LIN {X 0,Y 229.881,Z 707.672,A -85,B 0,C 180,E1 18522.942,E2 18522.942} C_VEL
LIN {X 0,Y 219.787,Z 692.83,A -85,B 0,C 180,E1 18532.814,E2 18532.814} C_VEL
LIN {X 0,Y 216.268,Z 686.361,A -85,B 0,C 180,E1 18540.004,E2 18540.004} C_VEL
LIN {X 0,Y 217.024,Z 688.955,A -85,B 0,C 180,E1 18552.29,E2 18552.29} C_VEL
LIN {X 0,Y 226.193,Z 701.763,A -85,B 0,C 180,E1 18563.446,E2 18563.446} C_VEL
LIN {X 0,Y 243.494,Z 730.82,A -85,B 0,C 180,E1 18574.667,E2 18574.667} C_VEL
LIN {X 0,Y 255.556,Z 766.15,A -85,B 0,C 180,E1 18582.726,E2 18582.726} C_VEL
LIN {X 0,Y 253.616,Z 779.963,A -85,B 0,C 180,E1 18584.484,E2 18584.484} C_VEL
LIN {X 0,Y 237.279,Z 822.45,A -85,B 0,C 180,E1 18590.836,E2 18590.836} C_VEL
LIN {X 0,Y 221.036,Z 856.867,A -85,B 0,C 180,E1 18601.276,E2 18601.276} C_VEL
LIN {X 0,Y 213.518,Z 876.846,A -85,B 0,C 180,E1 18613.662,E2 18613.662} C_VEL
LIN {X 0,Y 213.499,Z 883.891,A -85,B 0,C 180,E1 18623.879,E2 18623.879} C_VEL
LIN {X 0,Y 213.953,Z 882.641,A -85,B 0,C 180,E1 18634.067,E2 18634.067} C_VEL
LIN {X 0,Y 214.175,Z 868.105,A -85,B 0,C 180,E1 18646.928,E2 18646.928} C_VEL
LIN {X 0,Y 220.9,Z 839.18,A -85,B 0,C 180,E1 18658.743,E2 18658.743} C_VEL
LIN {X 0,Y 232.247,Z 798.241,A -85,B 0,C 180,E1 18667.481,E2 18667.481} C_VEL
LIN {X 0,Y 239.047,Z 758.866,A -85,B 0,C 180,E1 18672.107,E2 18672.107} C_VEL
LIN {X 0,Y 223.377,Z 710.425,A -85,B 0,C 180,E1 18677.976,E2 18677.976} C_VEL
LIN {X 0,Y 208.041,Z 678.81,A -85,B 0,C 180,E1 18682.787,E2 18682.787} C_VEL
LIN {X 0,Y 208.536,Z 678.81,A -85,B 0,C 180,E1 18696.401,E2 18696.401} C_VEL
LIN {X 0,Y 209.842,Z 678.81,A -85,B 0,C 180,E1 18709.579,E2 18709.579} C_VEL
LIN {X 0,Y 210.218,Z 678.81,A -85,B 0,C 180,E1 18722.064,E2 18722.064} C_VEL
LIN {X 0,Y 209.548,Z 678.81,A -85,B 0,C 180,E1 18734.679,E2 18734.679} C_VEL
LIN {X 0,Y 208.418,Z 678.81,A -85,B 0,C 180,E1 18748.378,E2 18748.378} C_VEL
LIN {X 0,Y 207.707,Z 678.81,A -85,B 0,C 180,E1 18757.847,E2 18757.847} C_VEL
LIN {X 0,Y 199.525,Z 678.81,A -85,B 0,C 180,E1 18767.645,E2 18767.645} C_VEL
LIN {X 0,Y 200.068,Z 678.81,A -85,B 0,C 180,E1 18780.723,E2 18780.723} C_VEL
LIN {X 0,Y 200.672,Z 680.538,A -85,B 0,C 180,E1 18786.541,E2 18786.541} C_VEL
LIN {X 0,Y 219.908,Z 721.807,A -85,B 0,C 180,E1 18793.945,E2 18793.945} C_VEL
LIN {X 0,Y 225.033,Z 755.949,A -85,B 0,C 180,E1 18800.294,E2 18800.294} C_VEL
LIN {X 0,Y 215.989,Z 790.154,A -85,B 0,C 180,E1 18808.49,E2 18808.49} C_VEL
LIN {X 0,Y 208.94,Z 812.982,A -85,B 0,C 180,E1 18819.406,E2 18819.406} C_VEL
LIN {X 0,Y 206.98,Z 821.875,A -85,B 0,C 180,E1 18829.265,E2 18829.265} C_VEL
LIN {X 0,Y 211.489,Z 820.688,A -85,B 0,C 180,E1 18842.559,E2 18842.559} C_VEL
LIN {X 0,Y 222.679,Z 806.166,A -85,B 0,C 180,E1 18853.748,E2 18853.748} C_VEL
LIN {X 0,Y 239.014,Z 776.963,A -85,B 0,C 180,E1 18862.905,E2 18862.905} C_VEL
LIN {X 0,Y 239.061,Z 749.813,A -85,B 0,C 180,E1 18870.717,E2 18870.717} C_VEL
LIN {X 0,Y 229.457,Z 720.051,A -85,B 0,C 180,E1 18881.194,E2 18881.194} C_VEL
LIN {X 0,Y 218.851,Z 700.999,A -85,B 0,C 180,E1 18892.533,E2 18892.533} C_VEL
LIN {X 0,Y 214.934,Z 694.204,A -85,B 0,C 180,E1 18901.016,E2 18901.016} C_VEL
LIN {X 0,Y 215.807,Z 696.88,A -85,B 0,C 180,E1 18911.921,E2 18911.921} C_VEL
LIN {X 0,Y 224.295,Z 709.472,A -85,B 0,C 180,E1 18922.88,E2 18922.88} C_VEL
LIN {X 0,Y 239.571,Z 737.112,A -85,B 0,C 180,E1 18933.939,E2 18933.939} C_VEL
LIN {X 0,Y 249.788,Z 770.735,A -85,B 0,C 180,E1 18942.009,E2 18942.009} C_VEL
LIN {X 0,Y 234.134,Z 815.138,A -85,B 0,C 180,E1 18948.201,E2 18948.201} C_VEL
LIN {X 0,Y 216.296,Z 851.412,A -85,B 0,C 180,E1 18958.25,E2 18958.25} C_VEL
LIN {X 0,Y 206.081,Z 874.611,A -85,B 0,C 180,E1 18971.855,E2 18971.855} C_VEL
LIN {X 0,Y 205.649,Z 883.042,A -85,B 0,C 180,E1 18985.094,E2 18985.094} C_VEL
LIN {X 0,Y 205.813,Z 879.931,A -85,B 0,C 180,E1 18996.35,E2 18996.35} C_VEL
LIN {X 0,Y 206.758,Z 862.386,A -85,B 0,C 180,E1 19009.844,E2 19009.844} C_VEL
LIN {X 0,Y 215.77,Z 829.843,A -85,B 0,C 180,E1 19021.836,E2 19021.836} C_VEL
LIN {X 0,Y 227.885,Z 786.903,A -85,B 0,C 180,E1 19029.909,E2 19029.909} C_VEL
LIN {X 0,Y 231.839,Z 760.664,A -85,B 0,C 180,E1 19032.91,E2 19032.91} C_VEL
LIN {X 0,Y 217.334,Z 714.047,A -85,B 0,C 180,E1 19038.986,E2 19038.986} C_VEL
LIN {X 0,Y 200.023,Z 678.81,A -85,B 0,C 180,E1 19044.727,E2 19044.727} C_VEL
LIN {X 0,Y 200.91,Z 678.81,A -85,B 0,C 180,E1 19060.764,E2 19060.764} C_VEL
LIN {X 0,Y 202.255,Z 678.81,A -85,B 0,C 180,E1 19073.533,E2 19073.533} C_VEL
LIN {X 0,Y 201.927,Z 678.81,A -85,B 0,C 180,E1 19086.469,E2 19086.469} C_VEL
LIN {X 0,Y 201.016,Z 678.81,A -85,B 0,C 180,E1 19099.856,E2 19099.856} C_VEL
LIN {X 0,Y 199.794,Z 678.81,A -85,B 0,C 180,E1 19114.724,E2 19114.724} C_VEL
LIN {X 0,Y 199.525,Z 678.81,A -85,B 0,C 180,E1 19127.645,E2 19127.645} C_VEL
LIN {X 0,Y 191.668,Z 678.81,A -85,B 0,C 180,E1 19137.868,E2 19137.868} C_VEL
LIN {X 0,Y 192.303,Z 680.013,A -85,B 0,C 180,E1 19144.277,E2 19144.277} C_VEL
LIN {X 0,Y 212.255,Z 721.579,A -85,B 0,C 180,E1 19152.421,E2 19152.421} C_VEL
LIN {X 0,Y 217.81,Z 755.571,A -85,B 0,C 180,E1 19159.042,E2 19159.042} C_VEL
LIN {X 0,Y 208.829,Z 789.974,A -85,B 0,C 180,E1 19167.397,E2 19167.397} C_VEL
LIN {X 0,Y 201.296,Z 813.354,A -85,B 0,C 180,E1 19178.589,E2 19178.589} C_VEL
LIN {X 0,Y 199.104,Z 823.33,A -85,B 0,C 180,E1 19190.059,E2 19190.059} C_VEL
LIN {X 0,Y 204.361,Z 821.543,A -85,B 0,C 180,E1 19203.844,E2 19203.844} C_VEL
LIN {X 0,Y 217.393,Z 805.196,A -85,B 0,C 180,E1 19215.88,E2 19215.88} C_VEL
LIN {X 0,Y 233.806,Z 774.97,A -85,B 0,C 180,E1 19225.119,E2 19225.119} C_VEL
LIN {X 0,Y 232.12,Z 746.503,A -85,B 0,C 180,E1 19234.176,E2 19234.176} C_VEL
LIN {X 0,Y 222.959,Z 720.424,A -85,B 0,C 180,E1 19245.089,E2 19245.089} C_VEL
LIN {X 0,Y 215.766,Z 706.799,A -85,B 0,C 180,E1 19255.213,E2 19255.213} C_VEL
LIN {X 0,Y 213.643,Z 701.951,A -85,B 0,C 180,E1 19262.04,E2 19262.04} C_VEL
LIN {X 0,Y 214.62,Z 705.005,A -85,B 0,C 180,E1 19271.73,E2 19271.73} C_VEL
LIN {X 0,Y 222.354,Z 717.478,A -85,B 0,C 180,E1 19282.508,E2 19282.508} C_VEL
LIN {X 0,Y 235.487,Z 743.318,A -85,B 0,C 180,E1 19293.22,E2 19293.22} C_VEL
LIN {X 0,Y 243.997,Z 775.784,A -85,B 0,C 180,E1 19301.391,E2 19301.391} C_VEL
LIN {X 0,Y 225.894,Z 819.243,A -85,B 0,C 180,E1 19307.758,E2 19307.758} C_VEL
LIN {X 0,Y 207.434,Z 854.096,A -85,B 0,C 180,E1 19318.584,E2 19318.584} C_VEL
LIN {X 0,Y 197.999,Z 874.565,A -85,B 0,C 180,E1 19332.096,E2 19332.096} C_VEL
LIN {X 0,Y 197.523,Z 881.59,A -85,B 0,C 180,E1 19343.382,E2 19343.382} C_VEL
LIN {X 0,Y 197.998,Z 879.68,A -85,B 0,C 180,E1 19354.942,E2 19354.942} C_VEL
LIN {X 0,Y 198.588,Z 863.33,A -85,B 0,C 180,E1 19369.163,E2 19369.163} C_VEL
LIN {X 0,Y 207.077,Z 833.12,A -85,B 0,C 180,E1 19381.476,E2 19381.476} C_VEL
LIN {X 0,Y 219.379,Z 791.904,A -85,B 0,C 180,E1 19390.105,E2 19390.105} C_VEL
LIN {X 0,Y 224.696,Z 762.234,A -85,B 0,C 180,E1 19393.787,E2 19393.787} C_VEL
LIN {X 0,Y 210.704,Z 716.189,A -85,B 0,C 180,E1 19400.235,E2 19400.235} C_VEL
LIN {X 0,Y 191.849,Z 678.81,A -85,B 0,C 180,E1 19406.993,E2 19406.993} C_VEL
LIN {X 0,Y 192.609,Z 678.81,A -85,B 0,C 180,E1 19419.228,E2 19419.228} C_VEL
LIN {X 0,Y 194.175,Z 678.81,A -85,B 0,C 180,E1 19433.263,E2 19433.263} C_VEL
LIN {X 0,Y 193.88,Z 678.81,A -85,B 0,C 180,E1 19446.738,E2 19446.738} C_VEL
LIN {X 0,Y 192.831,Z 678.81,A -85,B 0,C 180,E1 19460.737,E2 19460.737} C_VEL
LIN {X 0,Y 191.686,Z 678.81,A -85,B 0,C 180,E1 19476.421,E2 19476.421} C_VEL
LIN {X 0,Y 191.628,Z 678.81,A -85,B 0,C 180,E1 19493.563,E2 19493.563} C_VEL
LIN {X 0,Y 191.668,Z 678.81,A -85,B 0,C 180,E1 19497.868,E2 19497.868} C_VEL
LIN {X 0,Y 191.635,Z 685.766,A -85,B 0,C 180,E1 19502.561,E2 19502.561} C_VEL
LIN {X 0,Y 194.981,Z 698.935,A -85,B 0,C 180,E1 19506.133,E2 19506.133} C_VEL
LIN {X 0,Y 208.603,Z 735.9,A -85,B 0,C 180,E1 19513.694,E2 19513.694} C_VEL
LIN {X 0,Y 209.864,Z 765.32,A -85,B 0,C 180,E1 19519.915,E2 19519.915} C_VEL
LIN {X 0,Y 199.146,Z 798.07,A -85,B 0,C 180,E1 19529.344,E2 19529.344} C_VEL
LIN {X 0,Y 192.296,Z 818.117,A -85,B 0,C 180,E1 19541.379,E2 19541.379} C_VEL
LIN {X 0,Y 192.318,Z 825.544,A -85,B 0,C 180,E1 19555.721,E2 19555.721} C_VEL
LIN {X 0,Y 201.587,Z 818.107,A -85,B 0,C 180,E1 19569.783,E2 19569.783} C_VEL
LIN {X 0,Y 217.802,Z 796.184,A -85,B 0,C 180,E1 19581.054,E2 19581.054} C_VEL
LIN {X 0,Y 227.781,Z 775.465,A -85,B 0,C 180,E1 19586.917,E2 19586.917} C_VEL
LIN {X 0,Y 226.105,Z 747.296,A -85,B 0,C 180,E1 19596.623,E2 19596.623} C_VEL
LIN {X 0,Y 217.743,Z 722.229,A -85,B 0,C 180,E1 19608.699,E2 19608.699} C_VEL
LIN {X 0,Y 212.516,Z 709.99,A -85,B 0,C 180,E1 19621.027,E2 19621.027} C_VEL
LIN {X 0,Y 213.137,Z 712.726,A -85,B 0,C 180,E1 19631.294,E2 19631.294} C_VEL
LIN {X 0,Y 220.191,Z 725.55,A -85,B 0,C 180,E1 19642.281,E2 19642.281} C_VEL
LIN {X 0,Y 231.93,Z 751.303,A -85,B 0,C 180,E1 19653.122,E2 19653.122} C_VEL
LIN {X 0,Y 237.549,Z 778.975,A -85,B 0,C 180,E1 19660.291,E2 19660.291} C_VEL
LIN {X 0,Y 218.507,Z 821.527,A -85,B 0,C 180,E1 19666.952,E2 19666.952} C_VEL
LIN {X 0,Y 199.834,Z 854.414,A -85,B 0,C 180,E1 19677.887,E2 19677.887} C_VEL
LIN {X 0,Y 190.206,Z 873.601,A -85,B 0,C 180,E1 19691.389,E2 19691.389} C_VEL
LIN {X 0,Y 190.024,Z 880.843,A -85,B 0,C 180,E1 19706.756,E2 19706.756} C_VEL
LIN {X 0,Y 189.875,Z 877.181,A -85,B 0,C 180,E1 19716.885,E2 19716.885} C_VEL
LIN {X 0,Y 191.335,Z 858.875,A -85,B 0,C 180,E1 19731.52,E2 19731.52} C_VEL
LIN {X 0,Y 201.289,Z 827.068,A -85,B 0,C 180,E1 19743.78,E2 19743.78} C_VEL
LIN {X 0,Y 214.537,Z 783.538,A -85,B 0,C 180,E1 19752.221,E2 19752.221} C_VEL
LIN {X 0,Y 217.438,Z 763.356,A -85,B 0,C 180,E1 19754.787,E2 19754.787} C_VEL
LIN {X 0,Y 203.878,Z 717.945,A -85,B 0,C 180,E1 19761.652,E2 19761.652} C_VEL
LIN {X 0,Y 183.912,Z 678.81,A -85,B 0,C 180,E1 19769.058,E2 19769.058} C_VEL
LIN {X 0,Y 184.914,Z 678.81,A -85,B 0,C 180,E1 19783.301,E2 19783.301} C_VEL
LIN {X 0,Y 186.823,Z 678.81,A -85,B 0,C 180,E1 19797.667,E2 19797.667} C_VEL
LIN {X 0,Y 185.641,Z 678.81,A -85,B 0,C 180,E1 19811.788,E2 19811.788} C_VEL
LIN {X 0,Y 184.161,Z 678.81,A -85,B 0,C 180,E1 19826.947,E2 19826.947} C_VEL
LIN {X 0,Y 183.344,Z 678.81,A -85,B 0,C 180,E1 19844.709,E2 19844.709} C_VEL
LIN {X 0,Y 184.123,Z 680.189,A -85,B 0,C 180,E1 19861.813,E2 19861.813} C_VEL
LIN {X 0,Y 194.981,Z 698.935,A -85,B 0,C 180,E1 19866.133,E2 19866.133} C_VEL
LIN {X 0,Y 199.908,Z 730.202,A -85,B 0,C 180,E1 19870.917,E2 19870.917} C_VEL
LIN {X 0,Y 203.53,Z 761.737,A -85,B 0,C 180,E1 19877.89,E2 19877.89} C_VEL
LIN {X 0,Y 192.743,Z 795.512,A -85,B 0,C 180,E1 19887.18,E2 19887.18} C_VEL
LIN {X 0,Y 184.723,Z 818.218,A -85,B 0,C 180,E1 19900.236,E2 19900.236} C_VEL
LIN {X 0,Y 183.458,Z 826.079,A -85,B 0,C 180,E1 19911.854,E2 19911.854} C_VEL
LIN {X 0,Y 190.502,Z 823.157,A -85,B 0,C 180,E1 19926.688,E2 19926.688} C_VEL
LIN {X 0,Y 205.895,Z 805.593,A -85,B 0,C 180,E1 19939.301,E2 19939.301} C_VEL
LIN {X 0,Y 221.461,Z 779.214,A -85,B 0,C 180,E1 19947.714,E2 19947.714} C_VEL
LIN {X 0,Y 221.211,Z 753.146,A -85,B 0,C 180,E1 19957.251,E2 19957.251} C_VEL
LIN {X 0,Y 215.046,Z 729.857,A -85,B 0,C 180,E1 19968.814,E2 19968.814} C_VEL
LIN {X 0,Y 210.827,Z 717.776,A -85,B 0,C 180,E1 19981.035,E2 19981.035} C_VEL
LIN {X 0,Y 211.345,Z 720.576,A -85,B 0,C 180,E1 19991.042,E2 19991.042} C_VEL
LIN {X 0,Y 217.754,Z 733.517,A -85,B 0,C 180,E1 20002.141,E2 20002.141} C_VEL
LIN {X 0,Y 227.73,Z 758.407,A -85,B 0,C 180,E1 20012.79,E2 20012.79} C_VEL
LIN {X 0,Y 231.047,Z 782.48,A -85,B 0,C 180,E1 20019.164,E2 20019.164} C_VEL
LIN {X 0,Y 210.833,Z 824.25,A -85,B 0,C 180,E1 20026.249,E2 20026.249} C_VEL
LIN {X 0,Y 190.974,Z 856.722,A -85,B 0,C 180,E1 20038.234,E2 20038.234} C_VEL
LIN {X 0,Y 181.452,Z 875.348,A -85,B 0,C 180,E1 20054.138,E2 20054.138} C_VEL
LIN {X 0,Y 182.323,Z 879.653,A -85,B 0,C 180,E1 20067.615,E2 20067.615} C_VEL
LIN {X 0,Y 181.577,Z 872.771,A -85,B 0,C 180,E1 20080.839,E2 20080.839} C_VEL
LIN {X 0,Y 185.763,Z 850.113,A -85,B 0,C 180,E1 20096.014,E2 20096.014} C_VEL
LIN {X 0,Y 198.033,Z 814.084,A -85,B 0,C 180,E1 20107.81,E2 20107.81} C_VEL
LIN {X 0,Y 210.974,Z 768.884,A -85,B 0,C 180,E1 20115.096,E2 20115.096} C_VEL
LIN {X 0,Y 198.838,Z 723.531,A -85,B 0,C 180,E1 20122.478,E2 20122.478} C_VEL
LIN {X 0,Y 175.983,Z 678.81,A -85,B 0,C 180,E1 20132.539,E2 20132.539} C_VEL
LIN {X 0,Y 177.584,Z 678.81,A -85,B 0,C 180,E1 20149.337,E2 20149.337} C_VEL
LIN {X 0,Y 178.102,Z 678.81,A -85,B 0,C 180,E1 20162.437,E2 20162.437} C_VEL
LIN {X 0,Y 177.02,Z 678.81,A -85,B 0,C 180,E1 20177.456,E2 20177.456} C_VEL
LIN {X 0,Y 175.448,Z 678.81,A -85,B 0,C 180,E1 20194.744,E2 20194.744} C_VEL
LIN {X 0,Y 175.163,Z 678.81,A -85,B 0,C 180,E1 20209.476,E2 20209.476} C_VEL
LIN {X 0,Y 175.879,Z 680.501,A -85,B 0,C 180,E1 20218.99,E2 20218.99} C_VEL
LIN {X 0,Y 196.233,Z 718.883,A -85,B 0,C 180,E1 20228.459,E2 20228.459} C_VEL
LIN {X 0,Y 199.908,Z 730.202,A -85,B 0,C 180,E1 20230.917,E2 20230.917} C_VEL
LIN {X 0,Y 196.606,Z 760.663,A -85,B 0,C 180,E1 20236.252,E2 20236.252} C_VEL
LIN {X 0,Y 185.716,Z 795.329,A -85,B 0,C 180,E1 20245.9,E2 20245.9} C_VEL
LIN {X 0,Y 176.984,Z 818.89,A -85,B 0,C 180,E1 20259.587,E2 20259.587} C_VEL
LIN {X 0,Y 176.303,Z 827.866,A -85,B 0,C 180,E1 20275.343,E2 20275.343} C_VEL
LIN {X 0,Y 186.15,Z 821.865,A -85,B 0,C 180,E1 20290.703,E2 20290.703} C_VEL
LIN {X 0,Y 204.148,Z 800.993,A -85,B 0,C 180,E1 20303.031,E2 20303.031} C_VEL
LIN {X 0,Y 215.458,Z 781.062,A -85,B 0,C 180,E1 20309.253,E2 20309.253} C_VEL
LIN {X 0,Y 215.942,Z 756.697,A -85,B 0,C 180,E1 20318.839,E2 20318.839} C_VEL
LIN {X 0,Y 211.112,Z 735.388,A -85,B 0,C 180,E1 20330.696,E2 20330.696} C_VEL
LIN {X 0,Y 208.624,Z 725.403,A -85,B 0,C 180,E1 20342.089,E2 20342.089} C_VEL
LIN {X 0,Y 209.224,Z 728.445,A -85,B 0,C 180,E1 20350.928,E2 20350.928} C_VEL
LIN {X 0,Y 214.799,Z 740.892,A -85,B 0,C 180,E1 20361.777,E2 20361.777} C_VEL
LIN {X 0,Y 223.39,Z 766.243,A -85,B 0,C 180,E1 20372.742,E2 20372.742} C_VEL
LIN {X 0,Y 224.629,Z 785.836,A -85,B 0,C 180,E1 20377.998,E2 20377.998} C_VEL
LIN {X 0,Y 203.085,Z 826.997,A -85,B 0,C 180,E1 20385.529,E2 20385.529} C_VEL
LIN {X 0,Y 183.402,Z 856.858,A -85,B 0,C 180,E1 20397.463,E2 20397.463} C_VEL
LIN {X 0,Y 173.541,Z 874.524,A -85,B 0,C 180,E1 20413.836,E2 20413.836} C_VEL
LIN {X 0,Y 174.354,Z 878.411,A -85,B 0,C 180,E1 20427.506,E2 20427.506} C_VEL
LIN {X 0,Y 173.696,Z 872.396,A -85,B 0,C 180,E1 20440.063,E2 20440.063} C_VEL
LIN {X 0,Y 177.216,Z 851.594,A -85,B 0,C 180,E1 20455.496,E2 20455.496} C_VEL
LIN {X 0,Y 189.579,Z 817.024,A -85,B 0,C 180,E1 20467.979,E2 20467.979} C_VEL
LIN {X 0,Y 203.916,Z 771.307,A -85,B 0,C 180,E1 20475.914,E2 20475.914} C_VEL
LIN {X 0,Y 192.92,Z 727.271,A -85,B 0,C 180,E1 20483.663,E2 20483.663} C_VEL
LIN {X 0,Y 170.756,Z 684.849,A -85,B 0,C 180,E1 20493.427,E2 20493.427} C_VEL
LIN {X 0,Y 168.031,Z 678.81,A -85,B 0,C 180,E1 20495.411,E2 20495.411} C_VEL
LIN {X 0,Y 169.908,Z 678.81,A -85,B 0,C 180,E1 20512.295,E2 20512.295} C_VEL
LIN {X 0,Y 170.083,Z 678.81,A -85,B 0,C 180,E1 20522.552,E2 20522.552} C_VEL
LIN {X 0,Y 168.667,Z 678.81,A -85,B 0,C 180,E1 20539.141,E2 20539.141} C_VEL
LIN {X 0,Y 167.217,Z 678.81,A -85,B 0,C 180,E1 20556.145,E2 20556.145} C_VEL
LIN {X 0,Y 167.14,Z 678.81,A -85,B 0,C 180,E1 20573.831,E2 20573.831} C_VEL
LIN {X 0,Y 167.925,Z 681.626,A -85,B 0,C 180,E1 20575.923,E2 20575.923} C_VEL
LIN {X 0,Y 187.694,Z 716.2,A -85,B 0,C 180,E1 20585.858,E2 20585.858} C_VEL
LIN {X 0,Y 196.478,Z 750.492,A -85,B 0,C 180,E1 20593.869,E2 20593.869} C_VEL
LIN {X 0,Y 196.606,Z 760.663,A -85,B 0,C 180,E1 20596.252,E2 20596.252} C_VEL
LIN {X 0,Y 181.741,Z 787.468,A -85,B 0,C 180,E1 20601.78,E2 20601.78} C_VEL
LIN {X 0,Y 170.876,Z 814.989,A -85,B 0,C 180,E1 20615.095,E2 20615.095} C_VEL
LIN {X 0,Y 167.385,Z 826.908,A -85,B 0,C 180,E1 20628.501,E2 20628.501} C_VEL
LIN {X 0,Y 172.888,Z 827.721,A -85,B 0,C 180,E1 20644.788,E2 20644.788} C_VEL
LIN {X 0,Y 187.531,Z 814.98,A -85,B 0,C 180,E1 20658.462,E2 20658.462} C_VEL
LIN {X 0,Y 208.514,Z 787.522,A -85,B 0,C 180,E1 20669.038,E2 20669.038} C_VEL
LIN {X 0,Y 210.916,Z 762.499,A -85,B 0,C 180,E1 20679.47,E2 20679.47} C_VEL
LIN {X 0,Y 207.647,Z 741.923,A -85,B 0,C 180,E1 20691.597,E2 20691.597} C_VEL
LIN {X 0,Y 206.242,Z 733.037,A -85,B 0,C 180,E1 20702.113,E2 20702.113} C_VEL
LIN {X 0,Y 206.72,Z 735.941,A -85,B 0,C 180,E1 20710.58,E2 20710.58} C_VEL
LIN {X 0,Y 212.681,Z 750.912,A -85,B 0,C 180,E1 20723.112,E2 20723.112} C_VEL
LIN {X 0,Y 219.069,Z 776.779,A -85,B 0,C 180,E1 20733.661,E2 20733.661} C_VEL
LIN {X 0,Y 218.631,Z 788.225,A -85,B 0,C 180,E1 20736.661,E2 20736.661} C_VEL
LIN {X 0,Y 196.277,Z 828.113,A -85,B 0,C 180,E1 20744.342,E2 20744.342} C_VEL
LIN {X 0,Y 175.18,Z 857.887,A -85,B 0,C 180,E1 20757.219,E2 20757.219} C_VEL
LIN {X 0,Y 165.466,Z 874.215,A -85,B 0,C 180,E1 20774.395,E2 20774.395} C_VEL
LIN {X 0,Y 166.403,Z 877.163,A -85,B 0,C 180,E1 20787.386,E2 20787.386} C_VEL
LIN {X 0,Y 165.732,Z 870.942,A -85,B 0,C 180,E1 20800.552,E2 20800.552} C_VEL
LIN {X 0,Y 170.234,Z 848.849,A -85,B 0,C 180,E1 20817.132,E2 20817.132} C_VEL
LIN {X 0,Y 183.552,Z 813.223,A -85,B 0,C 180,E1 20829.847,E2 20829.847} C_VEL
LIN {X 0,Y 196.383,Z 769.328,A -85,B 0,C 180,E1 20837.624,E2 20837.624} C_VEL
LIN {X 0,Y 185.101,Z 726.088,A -85,B 0,C 180,E1 20845.861,E2 20845.861} C_VEL
LIN {X 0,Y 163.425,Z 685.316,A -85,B 0,C 180,E1 20856.567,E2 20856.567} C_VEL
LIN {X 0,Y 160.189,Z 678.81,A -85,B 0,C 180,E1 20859.184,E2 20859.184} C_VEL
LIN {X 0,Y 162.627,Z 678.81,A -85,B 0,C 180,E1 20877.32,E2 20877.32} C_VEL
LIN {X 0,Y 161.203,Z 678.81,A -85,B 0,C 180,E1 20893.607,E2 20893.607} C_VEL
LIN {X 0,Y 159.404,Z 678.81,A -85,B 0,C 180,E1 20911.57,E2 20911.57} C_VEL
LIN {X 0,Y 159.077,Z 678.81,A -85,B 0,C 180,E1 20930.803,E2 20930.803} C_VEL
LIN {X 0,Y 180.251,Z 716.053,A -85,B 0,C 180,E1 20943.611,E2 20943.611} C_VEL
LIN {X 0,Y 189.374,Z 750.675,A -85,B 0,C 180,E1 20952.272,E2 20952.272} C_VEL
LIN {X 0,Y 187.091,Z 773.601,A -85,B 0,C 180,E1 20957.919,E2 20957.919} C_VEL
LIN {X 0,Y 181.741,Z 787.468,A -85,B 0,C 180,E1 20961.78,E2 20961.78} C_VEL
LIN {X 0,Y 166.207,Z 808.669,A -85,B 0,C 180,E1 20969.666,E2 20969.666} C_VEL
LIN {X 0,Y 159.577,Z 826.639,A -85,B 0,C 180,E1 20986.041,E2 20986.041} C_VEL
LIN {X 0,Y 162.555,Z 830.166,A -85,B 0,C 180,E1 21000.895,E2 21000.895} C_VEL
LIN {X 0,Y 176.753,Z 820.45,A -85,B 0,C 180,E1 21016.868,E2 21016.868} C_VEL
LIN {X 0,Y 197.463,Z 797.162,A -85,B 0,C 180,E1 21028.337,E2 21028.337} C_VEL
LIN {X 0,Y 203.893,Z 784.648,A -85,B 0,C 180,E1 21032.698,E2 21032.698} C_VEL
LIN {X 0,Y 205.599,Z 762.892,A -85,B 0,C 180,E1 21042.831,E2 21042.831} C_VEL
LIN {X 0,Y 203.597,Z 745.412,A -85,B 0,C 180,E1 21055.294,E2 21055.294} C_VEL
LIN {X 0,Y 203.51,Z 740.566,A -85,B 0,C 180,E1 21062.141,E2 21062.141} C_VEL
LIN {X 0,Y 204.481,Z 745.404,A -85,B 0,C 180,E1 21072.87,E2 21072.87} C_VEL
LIN {X 0,Y 210.18,Z 762.529,A -85,B 0,C 180,E1 21085.146,E2 21085.146} C_VEL
LIN {X 0,Y 213.921,Z 787.913,A -85,B 0,C 180,E1 21094.892,E2 21094.892} C_VEL
LIN {X 0,Y 189.96,Z 828.652,A -85,B 0,C 180,E1 21102.905,E2 21102.905} C_VEL
LIN {X 0,Y 168.365,Z 857.061,A -85,B 0,C 180,E1 21115.713,E2 21115.713} C_VEL
LIN {X 0,Y 157.644,Z 873.134,A -85,B 0,C 180,E1 21133.599,E2 21133.599} C_VEL
LIN {X 0,Y 158.437,Z 875.91,A -85,B 0,C 180,E1 21147.255,E2 21147.255} C_VEL
LIN {X 0,Y 157.773,Z 869.472,A -85,B 0,C 180,E1 21161.091,E2 21161.091} C_VEL
LIN {X 0,Y 163.032,Z 846.606,A -85,B 0,C 180,E1 21178.586,E2 21178.586} C_VEL
LIN {X 0,Y 177.32,Z 810.55,A -85,B 0,C 180,E1 21191.549,E2 21191.549} C_VEL
LIN {X 0,Y 189.271,Z 770.081,A -85,B 0,C 180,E1 21198.924,E2 21198.924} C_VEL
LIN {X 0,Y 178.682,Z 728.066,A -85,B 0,C 180,E1 21207.572,E2 21207.572} C_VEL
LIN {X 0,Y 159.045,Z 690.923,A -85,B 0,C 180,E1 21218.293,E2 21218.293} C_VEL
LIN {X 0,Y 152.534,Z 678.81,A -85,B 0,C 180,E1 21223.511,E2 21223.511} C_VEL
LIN {X 0,Y 154.552,Z 678.81,A -85,B 0,C 180,E1 21237.18,E2 21237.18} C_VEL
LIN {X 0,Y 153.015,Z 678.81,A -85,B 0,C 180,E1 21254.351,E2 21254.351} C_VEL
LIN {X 0,Y 151.206,Z 678.81,A -85,B 0,C 180,E1 21273.499,E2 21273.499} C_VEL
LIN {X 0,Y 151.189,Z 680.403,A -85,B 0,C 180,E1 21287.079,E2 21287.079} C_VEL
LIN {X 0,Y 171.8,Z 713.859,A -85,B 0,C 180,E1 21300.414,E2 21300.414} C_VEL
LIN {X 0,Y 181.997,Z 747.748,A -85,B 0,C 180,E1 21309.765,E2 21309.765} C_VEL
LIN {X 0,Y 180.729,Z 773.086,A -85,B 0,C 180,E1 21316.34,E2 21316.34} C_VEL
LIN {X 0,Y 168.083,Z 804.5,A -85,B 0,C 180,E1 21327.413,E2 21327.413} C_VEL
LIN {X 0,Y 166.207,Z 808.669,A -85,B 0,C 180,E1 21329.666,E2 21329.666} C_VEL
LIN {X 0,Y 152.821,Z 823.544,A -85,B 0,C 180,E1 21340.231,E2 21340.231} C_VEL
LIN {X 0,Y 152.821,Z 831.345,A -85,B 0,C 180,E1 21356.543,E2 21356.543} C_VEL
LIN {X 0,Y 164.559,Z 826.216,A -85,B 0,C 180,E1 21373.761,E2 21373.761} C_VEL
LIN {X 0,Y 185.302,Z 806.737,A -85,B 0,C 180,E1 21387.081,E2 21387.081} C_VEL
LIN {X 0,Y 197.267,Z 790.25,A -85,B 0,C 180,E1 21392.88,E2 21392.88} C_VEL
LIN {X 0,Y 200.645,Z 768.73,A -85,B 0,C 180,E1 21403.486,E2 21403.486} C_VEL
LIN {X 0,Y 200.057,Z 752.488,A -85,B 0,C 180,E1 21415.654,E2 21415.654} C_VEL
LIN {X 0,Y 200.429,Z 747.98,A -85,B 0,C 180,E1 21422.174,E2 21422.174} C_VEL
LIN {X 0,Y 201.771,Z 753.777,A -85,B 0,C 180,E1 21434.154,E2 21434.154} C_VEL
LIN {X 0,Y 206.595,Z 773.47,A -85,B 0,C 180,E1 21446.786,E2 21446.786} C_VEL
LIN {X 0,Y 206.872,Z 792.921,A -85,B 0,C 180,E1 21453.782,E2 21453.782} C_VEL
LIN {X 0,Y 181.428,Z 832.205,A -85,B 0,C 180,E1 21462.358,E2 21462.358} C_VEL
LIN {X 0,Y 158.801,Z 859.577,A -85,B 0,C 180,E1 21476.668,E2 21476.668} C_VEL
LIN {X 0,Y 149.46,Z 873.058,A -85,B 0,C 180,E1 21495.295,E2 21495.295} C_VEL
LIN {X 0,Y 150.471,Z 874.655,A -85,B 0,C 180,E1 21507.109,E2 21507.109} C_VEL
LIN {X 0,Y 149.828,Z 867.952,A -85,B 0,C 180,E1 21521.687,E2 21521.687} C_VEL
LIN {X 0,Y 155.386,Z 845.782,A -85,B 0,C 180,E1 21539.409,E2 21539.409} C_VEL
LIN {X 0,Y 170.294,Z 810.093,A -85,B 0,C 180,E1 21552.803,E2 21552.803} C_VEL
LIN {X 0,Y 182.334,Z 771.872,A -85,B 0,C 180,E1 21560.099,E2 21560.099} C_VEL
LIN {X 0,Y 172.489,Z 730.313,A -85,B 0,C 180,E1 21569.351,E2 21569.351} C_VEL
LIN {X 0,Y 152.994,Z 692.468,A -85,B 0,C 180,E1 21581.467,E2 21581.467} C_VEL
LIN {X 0,Y 145.199,Z 678.81,A -85,B 0,C 180,E1 21589.454,E2 21589.454} C_VEL
LIN {X 0,Y 145.952,Z 678.81,A -85,B 0,C 180,E1 21602.974,E2 21602.974} C_VEL
LIN {X 0,Y 144.067,Z 678.81,A -85,B 0,C 180,E1 21621.629,E2 21621.629} C_VEL
LIN {X 0,Y 143.061,Z 680.494,A -85,B 0,C 180,E1 21640.964,E2 21640.964} C_VEL
LIN {X 0,Y 162.247,Z 709.493,A -85,B 0,C 180,E1 21655.977,E2 21655.977} C_VEL
LIN {X 0,Y 174.073,Z 742.255,A -85,B 0,C 180,E1 21666.254,E2 21666.254} C_VEL
LIN {X 0,Y 175.196,Z 770.457,A -85,B 0,C 180,E1 21674.184,E2 21674.184} C_VEL
LIN {X 0,Y 161.606,Z 803.161,A -85,B 0,C 180,E1 21685.287,E2 21685.287} C_VEL
LIN {X 0,Y 152.821,Z 823.544,A -85,B 0,C 180,E1 21700.231,E2 21700.231} C_VEL
LIN {X 0,Y 144.011,Z 831.623,A -85,B 0,C 180,E1 21713.154,E2 21713.154} C_VEL
LIN {X 0,Y 152.68,Z 830.514,A -85,B 0,C 180,E1 21730.246,E2 21730.246} C_VEL
LIN {X 0,Y 171.92,Z 815.958,A -85,B 0,C 180,E1 21744.991,E2 21744.991} C_VEL
LIN {X 0,Y 191.227,Z 793.462,A -85,B 0,C 180,E1 21754.125,E2 21754.125} C_VEL
LIN {X 0,Y 195.65,Z 772.677,A -85,B 0,C 180,E1 21765.289,E2 21765.289} C_VEL
LIN {X 0,Y 196.344,Z 758.051,A -85,B 0,C 180,E1 21777.907,E2 21777.907} C_VEL
LIN {X 0,Y 197.26,Z 755.646,A -85,B 0,C 180,E1 21786.631,E2 21786.631} C_VEL
LIN {X 0,Y 199.737,Z 768.389,A -85,B 0,C 180,E1 21799.998,E2 21799.998} C_VEL
LIN {X 0,Y 202.27,Z 790.567,A -85,B 0,C 180,E1 21810.91,E2 21810.91} C_VEL
LIN {X 0,Y 197.43,Z 801.444,A -85,B 0,C 180,E1 21813.194,E2 21813.194} C_VEL
LIN {X 0,Y 170.648,Z 838.153,A -85,B 0,C 180,E1 21822.806,E2 21822.806} C_VEL
LIN {X 0,Y 148.068,Z 862.94,A -85,B 0,C 180,E1 21839.176,E2 21839.176} C_VEL
LIN {X 0,Y 141.533,Z 873.314,A -85,B 0,C 180,E1 21860.745,E2 21860.745} C_VEL
LIN {X 0,Y 142.668,Z 871.882,A -85,B 0,C 180,E1 21873.048,E2 21873.048} C_VEL
LIN {X 0,Y 143.315,Z 857.279,A -85,B 0,C 180,E1 21891.753,E2 21891.753} C_VEL
LIN {X 0,Y 155.541,Z 827.55,A -85,B 0,C 180,E1 21908.461,E2 21908.461} C_VEL
LIN {X 0,Y 172.339,Z 786.587,A -85,B 0,C 180,E1 21919.077,E2 21919.077} C_VEL
LIN {X 0,Y 175.133,Z 770.417,A -85,B 0,C 180,E1 21922.081,E2 21922.081} C_VEL
LIN {X 0,Y 165.307,Z 729.682,A -85,B 0,C 180,E1 21932.012,E2 21932.012} C_VEL
LIN {X 0,Y 147.928,Z 696.603,A -85,B 0,C 180,E1 21944.286,E2 21944.286} C_VEL
LIN {X 0,Y 138.131,Z 678.81,A -85,B 0,C 180,E1 21955.625,E2 21955.625} C_VEL
LIN {X 0,Y 137.322,Z 678.81,A -85,B 0,C 180,E1 21969.536,E2 21969.536} C_VEL
LIN {X 0,Y 135.85,Z 678.81,A -85,B 0,C 180,E1 21983.01,E2 21983.01} C_VEL
LIN {X 0,Y 135.146,Z 680.994,A -85,B 0,C 180,E1 21992.296,E2 21992.296} C_VEL
LIN {X 0,Y 145.957,Z 695.503,A -85,B 0,C 180,E1 22005.025,E2 22005.025} C_VEL
LIN {X 0,Y 161.762,Z 724.396,A -85,B 0,C 180,E1 22018.152,E2 22018.152} C_VEL
LIN {X 0,Y 169.174,Z 757.49,A -85,B 0,C 180,E1 22028.577,E2 22028.577} C_VEL
LIN {X 0,Y 165.6,Z 778.62,A -85,B 0,C 180,E1 22034.601,E2 22034.601} C_VEL
LIN {X 0,Y 151.321,Z 810.155,A -85,B 0,C 180,E1 22047.657,E2 22047.657} C_VEL
LIN {X 0,Y 143.779,Z 828.4,A -85,B 0,C 180,E1 22065.3,E2 22065.3} C_VEL
LIN {X 0,Y 144.011,Z 831.623,A -85,B 0,C 180,E1 22073.154,E2 22073.154} C_VEL
LIN {X 0,Y 142.125,Z 833.111,A -85,B 0,C 180,E1 22087.317,E2 22087.317} C_VEL
LIN {X 0,Y 160.385,Z 822.127,A -85,B 0,C 180,E1 22103.539,E2 22103.539} C_VEL
LIN {X 0,Y 185.34,Z 796.539,A -85,B 0,C 180,E1 22115.508,E2 22115.508} C_VEL
LIN {X 0,Y 190.553,Z 778.091,A -85,B 0,C 180,E1 22126.153,E2 22126.153} C_VEL
LIN {X 0,Y 192.337,Z 765.099,A -85,B 0,C 180,E1 22137.964,E2 22137.964} C_VEL
LIN {X 0,Y 193.505,Z 762.952,A -85,B 0,C 180,E1 22146.761,E2 22146.761} C_VEL
LIN {X 0,Y 195.503,Z 776.144,A -85,B 0,C 180,E1 22160.451,E2 22160.451} C_VEL
LIN {X 0,Y 196.439,Z 795.416,A -85,B 0,C 180,E1 22170.149,E2 22170.149} C_VEL
LIN {X 0,Y 168.637,Z 833.716,A -85,B 0,C 180,E1 22179.254,E2 22179.254} C_VEL
LIN {X 0,Y 143.82,Z 859.29,A -85,B 0,C 180,E1 22194.525,E2 22194.525} C_VEL
LIN {X 0,Y 133.618,Z 871.152,A -85,B 0,C 180,E1 22214.915,E2 22214.915} C_VEL
LIN {X 0,Y 134.512,Z 872.138,A -85,B 0,C 180,E1 22226.766,E2 22226.766} C_VEL
LIN {X 0,Y 133.963,Z 866.159,A -85,B 0,C 180,E1 22241.351,E2 22241.351} C_VEL
LIN {X 0,Y 139.971,Z 844.645,A -85,B 0,C 180,E1 22260.996,E2 22260.996} C_VEL
LIN {X 0,Y 156.536,Z 809.035,A -85,B 0,C 180,E1 22275.641,E2 22275.641} C_VEL
LIN {X 0,Y 168.54,Z 774.571,A -85,B 0,C 180,E1 22282.872,E2 22282.872} C_VEL
LIN {X 0,Y 160.422,Z 735.105,A -85,B 0,C 180,E1 22293.191,E2 22293.191} C_VEL
LIN {X 0,Y 144.906,Z 702.967,A -85,B 0,C 180,E1 22305.784,E2 22305.784} C_VEL
LIN {X 0,Y 134.295,Z 685.851,A -85,B 0,C 180,E1 22318.779,E2 22318.779} C_VEL
LIN {X 0,Y 129.401,Z 682.834,A -85,B 0,C 180,E1 22337.718,E2 22337.718} C_VEL
LIN {X 0,Y 133.708,Z 689.308,A -85,B 0,C 180,E1 22351.792,E2 22351.792} C_VEL
LIN {X 0,Y 144.426,Z 704.606,A -85,B 0,C 180,E1 22365.129,E2 22365.129} C_VEL
LIN {X 0,Y 157.645,Z 732.523,A -85,B 0,C 180,E1 22378.032,E2 22378.032} C_VEL
LIN {X 0,Y 162.683,Z 763.246,A -85,B 0,C 180,E1 22388.3,E2 22388.3} C_VEL
LIN {X 0,Y 157.089,Z 783.598,A -85,B 0,C 180,E1 22394.296,E2 22394.296} C_VEL
LIN {X 0,Y 142.385,Z 813.85,A -85,B 0,C 180,E1 22408.473,E2 22408.473} C_VEL
LIN {X 0,Y 135.761,Z 830.019,A -85,B 0,C 180,E1 22426.228,E2 22426.228} C_VEL
LIN {X 0,Y 142.125,Z 833.111,A -85,B 0,C 180,E1 22447.317,E2 22447.317} C_VEL
LIN {X 0,Y 147.733,Z 828.065,A -85,B 0,C 180,E1 22461.052,E2 22461.052} C_VEL
LIN {X 0,Y 173.484,Z 806.626,A -85,B 0,C 180,E1 22474.377,E2 22474.377} C_VEL
LIN {X 0,Y 180.773,Z 796.963,A -85,B 0,C 180,E1 22478.457,E2 22478.457} C_VEL
LIN {X 0,Y 186.256,Z 779.575,A -85,B 0,C 180,E1 22489.996,E2 22489.996} C_VEL
LIN {X 0,Y 189.153,Z 769.368,A -85,B 0,C 180,E1 22502.304,E2 22502.304} C_VEL
LIN {X 0,Y 189.841,Z 775.111,A -85,B 0,C 180,E1 22513.881,E2 22513.881} C_VEL
LIN {X 0,Y 191.041,Z 792.635,A -85,B 0,C 180,E1 22525.913,E2 22525.913} C_VEL
LIN {X 0,Y 189.03,Z 801.13,A -85,B 0,C 180,E1 22529.128,E2 22529.128} C_VEL
LIN {X 0,Y 160.021,Z 836.922,A -85,B 0,C 180,E1 22538.52,E2 22538.52} C_VEL
LIN {X 0,Y 134.237,Z 861.078,A -85,B 0,C 180,E1 22555.58,E2 22555.58} C_VEL
LIN {X 0,Y 125.567,Z 870.916,A -85,B 0,C 180,E1 22579.555,E2 22579.555} C_VEL
LIN {X 0,Y 126.728,Z 869.17,A -85,B 0,C 180,E1 22593.432,E2 22593.432} C_VEL
LIN {X 0,Y 128.12,Z 853.717,A -85,B 0,C 180,E1 22614.492,E2 22614.492} C_VEL
LIN {X 0,Y 141.893,Z 824.79,A -85,B 0,C 180,E1 22631.785,E2 22631.785} C_VEL
LIN {X 0,Y 160.496,Z 783.437,A -85,B 0,C 180,E1 22642.792,E2 22642.792} C_VEL
LIN {X 0,Y 159.44,Z 756.765,A -85,B 0,C 180,E1 22649.618,E2 22649.618} C_VEL
LIN {X 0,Y 148.376,Z 721.743,A -85,B 0,C 180,E1 22661.16,E2 22661.16} C_VEL
LIN {X 0,Y 134.895,Z 697.201,A -85,B 0,C 180,E1 22675.915,E2 22675.915} C_VEL
LIN {X 0,Y 129.387,Z 690.853,A -85,B 0,C 180,E1 22687.75,E2 22687.75} C_VEL
LIN {X 0,Y 131.392,Z 694.581,A -85,B 0,C 180,E1 22709.033,E2 22709.033} C_VEL
LIN {X 0,Y 142.959,Z 714.496,A -85,B 0,C 180,E1 22725.858,E2 22725.858} C_VEL
LIN {X 0,Y 153.559,Z 742.137,A -85,B 0,C 180,E1 22738.568,E2 22738.568} C_VEL
LIN {X 0,Y 155.709,Z 771.121,A -85,B 0,C 180,E1 22748.755,E2 22748.755} C_VEL
LIN {X 0,Y 139.688,Z 805.929,A -85,B 0,C 180,E1 22761.729,E2 22761.729} C_VEL
LIN {X 0,Y 128.871,Z 827.454,A -85,B 0,C 180,E1 22780.174,E2 22780.174} C_VEL
LIN {X 0,Y 130.697,Z 835.081,A -85,B 0,C 180,E1 22801.501,E2 22801.501} C_VEL
LIN {X 0,Y 147.733,Z 828.065,A -85,B 0,C 180,E1 22821.052,E2 22821.052} C_VEL
LIN {X 0,Y 159.407,Z 816.535,A -85,B 0,C 180,E1 22832.794,E2 22832.794} C_VEL
LIN {X 0,Y 174.264,Z 801.733,A -85,B 0,C 180,E1 22839.038,E2 22839.038} C_VEL
LIN {X 0,Y 180.922,Z 785.873,A -85,B 0,C 180,E1 22850.201,E2 22850.201} C_VEL
LIN {X 0,Y 184.731,Z 776.169,A -85,B 0,C 180,E1 22862.359,E2 22862.359} C_VEL
LIN {X 0,Y 185.254,Z 782.246,A -85,B 0,C 180,E1 22874.232,E2 22874.232} C_VEL
LIN {X 0,Y 185.265,Z 798.906,A -85,B 0,C 180,E1 22885.794,E2 22885.794} C_VEL
LIN {X 0,Y 180.531,Z 807.439,A -85,B 0,C 180,E1 22888.038,E2 22888.038} C_VEL
LIN {X 0,Y 149.968,Z 841.165,A -85,B 0,C 180,E1 22898.39,E2 22898.39} C_VEL
LIN {X 0,Y 124.72,Z 862.458,A -85,B 0,C 180,E1 22916.801,E2 22916.801} C_VEL
LIN {X 0,Y 117.601,Z 869.682,A -85,B 0,C 180,E1 22938.839,E2 22938.839} C_VEL
LIN {X 0,Y 118.742,Z 867.802,A -85,B 0,C 180,E1 22953.663,E2 22953.663} C_VEL
LIN {X 0,Y 120.626,Z 851.915,A -85,B 0,C 180,E1 22976.124,E2 22976.124} C_VEL
LIN {X 0,Y 136.137,Z 821.681,A -85,B 0,C 180,E1 22994.385,E2 22994.385} C_VEL
LIN {X 0,Y 155.185,Z 780.949,A -85,B 0,C 180,E1 23005.016,E2 23005.016} C_VEL
LIN {X 0,Y 149.764,Z 743.341,A -85,B 0,C 180,E1 23016.478,E2 23016.478} C_VEL
LIN {X 0,Y 137.626,Z 712.857,A -85,B 0,C 180,E1 23030.473,E2 23030.473} C_VEL
LIN {X 0,Y 130.389,Z 700.687,A -85,B 0,C 180,E1 23042.182,E2 23042.182} C_VEL
LIN {X 0,Y 127.47,Z 699.263,A -85,B 0,C 180,E1 23059.06,E2 23059.06} C_VEL
LIN {X 0,Y 131.557,Z 706.679,A -85,B 0,C 180,E1 23072.481,E2 23072.481} C_VEL
LIN {X 0,Y 140.905,Z 724.13,A -85,B 0,C 180,E1 23086.588,E2 23086.588} C_VEL
LIN {X 0,Y 148.75,Z 751.824,A -85,B 0,C 180,E1 23099.284,E2 23099.284} C_VEL
LIN {X 0,Y 147.726,Z 777.458,A -85,B 0,C 180,E1 23108.584,E2 23108.584} C_VEL
LIN {X 0,Y 130.373,Z 810.63,A -85,B 0,C 180,E1 23122.639,E2 23122.639} C_VEL
LIN {X 0,Y 120.307,Z 830.316,A -85,B 0,C 180,E1 23142.71,E2 23142.71} C_VEL
LIN {X 0,Y 123.584,Z 836.288,A -85,B 0,C 180,E1 23163.544,E2 23163.544} C_VEL
LIN {X 0,Y 141.965,Z 829.107,A -85,B 0,C 180,E1 23183.295,E2 23183.295} C_VEL
LIN {X 0,Y 159.407,Z 816.535,A -85,B 0,C 180,E1 23192.794,E2 23192.794} C_VEL
LIN {X 0,Y 167.631,Z 806.196,A -85,B 0,C 180,E1 23199.821,E2 23199.821} C_VEL
LIN {X 0,Y 175.735,Z 790.935,A -85,B 0,C 180,E1 23211.315,E2 23211.315} C_VEL
LIN {X 0,Y 180.006,Z 782.754,A -85,B 0,C 180,E1 23222.421,E2 23222.421} C_VEL
LIN {X 0,Y 180.309,Z 789.132,A -85,B 0,C 180,E1 23234.56,E2 23234.56} C_VEL
LIN {X 0,Y 178.828,Z 804.694,A -85,B 0,C 180,E1 23245.313,E2 23245.313} C_VEL
LIN {X 0,Y 148.112,Z 837.849,A -85,B 0,C 180,E1 23254.57,E2 23254.57} C_VEL
LIN {X 0,Y 119.446,Z 860.387,A -85,B 0,C 180,E1 23272.88,E2 23272.88} C_VEL
LIN {X 0,Y 109.653,Z 868.448,A -85,B 0,C 180,E1 23298.018,E2 23298.018} C_VEL
LIN {X 0,Y 110.767,Z 866.429,A -85,B 0,C 180,E1 23313.928,E2 23313.928} C_VEL
LIN {X 0,Y 113.298,Z 850.115,A -85,B 0,C 180,E1 23337.956,E2 23337.956} C_VEL
LIN {X 0,Y 129.963,Z 819.819,A -85,B 0,C 180,E1 23356.672,E2 23356.672} C_VEL
LIN {X 0,Y 148.538,Z 780.477,A -85,B 0,C 180,E1 23367.272,E2 23367.272} C_VEL
LIN {X 0,Y 143.885,Z 745.031,A -85,B 0,C 180,E1 23379.14,E2 23379.14} C_VEL
LIN {X 0,Y 133.578,Z 717.379,A -85,B 0,C 180,E1 23393.587,E2 23393.587} C_VEL
LIN {X 0,Y 128.403,Z 707.902,A -85,B 0,C 180,E1 23404.125,E2 23404.125} C_VEL
LIN {X 0,Y 126.528,Z 707.851,A -85,B 0,C 180,E1 23421.279,E2 23421.279} C_VEL
LIN {X 0,Y 131.754,Z 718.459,A -85,B 0,C 180,E1 23436.444,E2 23436.444} C_VEL
LIN {X 0,Y 140.713,Z 742.688,A -85,B 0,C 180,E1 23452.014,E2 23452.014} C_VEL
LIN {X 0,Y 143.054,Z 770.921,A -85,B 0,C 180,E1 23463.942,E2 23463.942} C_VEL
LIN {X 0,Y 134.289,Z 791.93,A -85,B 0,C 180,E1 23471.039,E2 23471.039} C_VEL
LIN {X 0,Y 117.836,Z 820.294,A -85,B 0,C 180,E1 23488.155,E2 23488.155} C_VEL
LIN {X 0,Y 111.958,Z 834.671,A -85,B 0,C 180,E1 23509.808,E2 23509.808} C_VEL
LIN {X 0,Y 121.825,Z 836.59,A -85,B 0,C 180,E1 23533.245,E2 23533.245} C_VEL
LIN {X 0,Y 146.707,Z 823.714,A -85,B 0,C 180,E1 23551.552,E2 23551.552} C_VEL
LIN {X 0,Y 167.631,Z 806.196,A -85,B 0,C 180,E1 23559.821,E2 23559.821} C_VEL
LIN {X 0,Y 169.942,Z 796.818,A -85,B 0,C 180,E1 23571.575,E2 23571.575} C_VEL
LIN {X 0,Y 174.973,Z 789.129,A -85,B 0,C 180,E1 23582.491,E2 23582.491} C_VEL
LIN {X 0,Y 174.995,Z 795.908,A -85,B 0,C 180,E1 23595.012,E2 23595.012} C_VEL
LIN {X 0,Y 172.639,Z 808.009,A -85,B 0,C 180,E1 23603.531,E2 23603.531} C_VEL
LIN {X 0,Y 139.445,Z 840.708,A -85,B 0,C 180,E1 23613.566,E2 23613.566} C_VEL
LIN {X 0,Y 111.345,Z 860.523,A -85,B 0,C 180,E1 23632.17,E2 23632.17} C_VEL
LIN {X 0,Y 101.722,Z 867.212,A -85,B 0,C 180,E1 23657.069,E2 23657.069} C_VEL
LIN {X 0,Y 102.767,Z 865.011,A -85,B 0,C 180,E1 23674.234,E2 23674.234} C_VEL
LIN {X 0,Y 106.11,Z 848.228,A -85,B 0,C 180,E1 23700.037,E2 23700.037} C_VEL
LIN {X 0,Y 124.813,Z 816.698,A -85,B 0,C 180,E1 23719.649,E2 23719.649} C_VEL
LIN {X 0,Y 142.002,Z 780.906,A -85,B 0,C 180,E1 23729.485,E2 23729.485} C_VEL
LIN {X 0,Y 137.94,Z 746.052,A -85,B 0,C 180,E1 23742.382,E2 23742.382} C_VEL
LIN {X 0,Y 129.509,Z 720.664,A -85,B 0,C 180,E1 23757.685,E2 23757.685} C_VEL
LIN {X 0,Y 125.308,Z 713.851,A -85,B 0,C 180,E1 23770.46,E2 23770.46} C_VEL
LIN {X 0,Y 126.574,Z 720.438,A -85,B 0,C 180,E1 23789.278,E2 23789.278} C_VEL
LIN {X 0,Y 132.996,Z 737.174,A -85,B 0,C 180,E1 23804.464,E2 23804.464} C_VEL
LIN {X 0,Y 137.187,Z 762.798,A -85,B 0,C 180,E1 23817.628,E2 23817.628} C_VEL
LIN {X 0,Y 134.157,Z 781.592,A -85,B 0,C 180,E1 23825.172,E2 23825.172} C_VEL
LIN {X 0,Y 115.568,Z 813.17,A -85,B 0,C 180,E1 23839.983,E2 23839.983} C_VEL
LIN {X 0,Y 104.417,Z 832.617,A -85,B 0,C 180,E1 23862.592,E2 23862.592} C_VEL
LIN {X 0,Y 109.938,Z 838.675,A -85,B 0,C 180,E1 23888.401,E2 23888.401} C_VEL
LIN {X 0,Y 132.524,Z 830.503,A -85,B 0,C 180,E1 23909.186,E2 23909.186} C_VEL
LIN {X 0,Y 162.82,Z 808.125,A -85,B 0,C 180,E1 23922.246,E2 23922.246} C_VEL
LIN {X 0,Y 169.942,Z 796.818,A -85,B 0,C 180,E1 23931.575,E2 23931.575} C_VEL
LIN {X 0,Y 169.963,Z 794.799,A -85,B 0,C 180,E1 23940.581,E2 23940.581} C_VEL
LIN {X 0,Y 169.577,Z 795.553,A -85,B 0,C 180,E1 23943.676,E2 23943.676} C_VEL
LIN {X 0,Y 169.4,Z 801.749,A -85,B 0,C 180,E1 23954.801,E2 23954.801} C_VEL
LIN {X 0,Y 166.77,Z 810.977,A -85,B 0,C 180,E1 23961.605,E2 23961.605} C_VEL
LIN {X 0,Y 131.929,Z 842.393,A -85,B 0,C 180,E1 23971.969,E2 23971.969} C_VEL
LIN {X 0,Y 101.737,Z 861.381,A -85,B 0,C 180,E1 23993.374,E2 23993.374} C_VEL
LIN {X 0,Y 94.529,Z 865.638,A -85,B 0,C 180,E1 24025.396,E2 24025.396} C_VEL
LIN {X 0,Y 94.354,Z 859.555,A -85,B 0,C 180,E1 24043.96,E2 24043.96} C_VEL
LIN {X 0,Y 105.138,Z 836.965,A -85,B 0,C 180,E1 24070.505,E2 24070.505} C_VEL
LIN {X 0,Y 127.331,Z 800.946,A -85,B 0,C 180,E1 24086.89,E2 24086.89} C_VEL
LIN {X 0,Y 135.614,Z 781.991,A -85,B 0,C 180,E1 24091.703,E2 24091.703} C_VEL
LIN {X 0,Y 132.698,Z 748.96,A -85,B 0,C 180,E1 24105.091,E2 24105.091} C_VEL
LIN {X 0,Y 126.052,Z 725.267,A -85,B 0,C 180,E1 24121.382,E2 24121.382} C_VEL
LIN {X 0,Y 122.851,Z 722.382,A -85,B 0,C 180,E1 24137.104,E2 24137.104} C_VEL
LIN {X 0,Y 125.324,Z 731.024,A -85,B 0,C 180,E1 24153.012,E2 24153.012} C_VEL
LIN {X 0,Y 130.531,Z 752.868,A -85,B 0,C 180,E1 24169.079,E2 24169.079} C_VEL
LIN {X 0,Y 129.863,Z 779.228,A -85,B 0,C 180,E1 24181.84,E2 24181.84} C_VEL
LIN {X 0,Y 109.603,Z 812.485,A -85,B 0,C 180,E1 24196.998,E2 24196.998} C_VEL
LIN {X 0,Y 96.668,Z 833.185,A -85,B 0,C 180,E1 24221.317,E2 24221.317} C_VEL
LIN {X 0,Y 103.445,Z 839.813,A -85,B 0,C 180,E1 24251.312,E2 24251.312} C_VEL
LIN {X 0,Y 128.391,Z 831.2,A -85,B 0,C 180,E1 24272.435,E2 24272.435} C_VEL
LIN {X 0,Y 158.215,Z 810.162,A -85,B 0,C 180,E1 24284.866,E2 24284.866} C_VEL
LIN {X 0,Y 165.732,Z 799.906,A -85,B 0,C 180,E1 24294.751,E2 24294.751} C_VEL
LIN {X 0,Y 169.577,Z 795.553,A -85,B 0,C 180,E1 24303.676,E2 24303.676} C_VEL
LIN {X 0,Y 163.409,Z 807.85,A -85,B 0,C 180,E1 24315.11,E2 24315.11} C_VEL
LIN {X 0,Y 160.587,Z 814.321,A -85,B 0,C 180,E1 24319.661,E2 24319.661} C_VEL
LIN {X 0,Y 123.471,Z 844.604,A -85,B 0,C 180,E1 24330.643,E2 24330.643} C_VEL
LIN {X 0,Y 95.27,Z 860.343,A -85,B 0,C 180,E1 24350.419,E2 24350.419} C_VEL
LIN {X 0,Y 86.531,Z 864.309,A -85,B 0,C 180,E1 24384.969,E2 24384.969} C_VEL
LIN {X 0,Y 86.486,Z 857.965,A -85,B 0,C 180,E1 24405.26,E2 24405.26} C_VEL
LIN {X 0,Y 99,Z 834.865,A -85,B 0,C 180,E1 24433.613,E2 24433.613} C_VEL
LIN {X 0,Y 122.564,Z 798.707,A -85,B 0,C 180,E1 24449.891,E2 24449.891} C_VEL
LIN {X 0,Y 129.367,Z 782.751,A -85,B 0,C 180,E1 24454.23,E2 24454.23} C_VEL
LIN {X 0,Y 127.903,Z 753.524,A -85,B 0,C 180,E1 24467.138,E2 24467.138} C_VEL
LIN {X 0,Y 123.5,Z 733.18,A -85,B 0,C 180,E1 24481.753,E2 24481.753} C_VEL
LIN {X 0,Y 121.337,Z 729.396,A -85,B 0,C 180,E1 24490.806,E2 24490.806} C_VEL
LIN {X 0,Y 121.309,Z 735.649,A -85,B 0,C 180,E1 24508.45,E2 24508.45} C_VEL
LIN {X 0,Y 124.902,Z 752.69,A -85,B 0,C 180,E1 24524.24,E2 24524.24} C_VEL
LIN {X 0,Y 124.611,Z 776.634,A -85,B 0,C 180,E1 24537.444,E2 24537.444} C_VEL
LIN {X 0,Y 117.473,Z 791.631,A -85,B 0,C 180,E1 24543.119,E2 24543.119} C_VEL
LIN {X 0,Y 96.559,Z 821.631,A -85,B 0,C 180,E1 24562.096,E2 24562.096} C_VEL
LIN {X 0,Y 88.153,Z 837.309,A -85,B 0,C 180,E1 24588.791,E2 24588.791} C_VEL
LIN {X 0,Y 98.411,Z 840.849,A -85,B 0,C 180,E1 24616.068,E2 24616.068} C_VEL
LIN {X 0,Y 127.253,Z 830.546,A -85,B 0,C 180,E1 24637.098,E2 24637.098} C_VEL
LIN {X 0,Y 153.199,Z 812.897,A -85,B 0,C 180,E1 24647.173,E2 24647.173} C_VEL
LIN {X 0,Y 162.098,Z 802.83,A -85,B 0,C 180,E1 24659.21,E2 24659.21} C_VEL
LIN {X 0,Y 163.97,Z 801.4,A -85,B 0,C 180,E1 24663.47,E2 24663.47} C_VEL
LIN {X 0,Y 163.409,Z 807.85,A -85,B 0,C 180,E1 24675.11,E2 24675.11} C_VEL
LIN {X 0,Y 155.405,Z 816.939,A -85,B 0,C 180,E1 24677.873,E2 24677.873} C_VEL
LIN {X 0,Y 148.086,Z 823.186,A -85,B 0,C 180,E1 24678.902,E2 24678.902} C_VEL
LIN {X 0,Y 110.788,Z 848.936,A -85,B 0,C 180,E1 24691.117,E2 24691.117} C_VEL
LIN {X 0,Y 83.939,Z 861.461,A -85,B 0,C 180,E1 24714.468,E2 24714.468} C_VEL
LIN {X 0,Y 78.711,Z 862.068,A -85,B 0,C 180,E1 24750,E2 24750} C_VEL
LIN {X 0,Y 81.383,Z 849.025,A -85,B 0,C 180,E1 24780.04,E2 24780.04} C_VEL
LIN {X 0,Y 102.279,Z 820.234,A -85,B 0,C 180,E1 24804.691,E2 24804.691} C_VEL
LIN {X 0,Y 123.101,Z 786.031,A -85,B 0,C 180,E1 24815.916,E2 24815.916} C_VEL
LIN {X 0,Y 123.106,Z 757.99,A -85,B 0,C 180,E1 24829.336,E2 24829.336} C_VEL
LIN {X 0,Y 120.353,Z 739.577,A -85,B 0,C 180,E1 24843.607,E2 24843.607} C_VEL
LIN {X 0,Y 117.962,Z 738.172,A -85,B 0,C 180,E1 24858.754,E2 24858.754} C_VEL
LIN {X 0,Y 119.344,Z 750.415,A -85,B 0,C 180,E1 24876.503,E2 24876.503} C_VEL
LIN {X 0,Y 119.814,Z 771.759,A -85,B 0,C 180,E1 24891.131,E2 24891.131} C_VEL
LIN {X 0,Y 115.798,Z 786.252,A -85,B 0,C 180,E1 24898.209,E2 24898.209} C_VEL
LIN {X 0,Y 92.75,Z 818.332,A -85,B 0,C 180,E1 24915.793,E2 24915.793} C_VEL
LIN {X 0,Y 80.235,Z 837.53,A -85,B 0,C 180,E1 24946.482,E2 24946.482} C_VEL
LIN {X 0,Y 91.446,Z 842.09,A -85,B 0,C 180,E1 24978.313,E2 24978.313} C_VEL
LIN {X 0,Y 121.488,Z 832.536,A -85,B 0,C 180,E1 24999.53,E2 24999.53} C_VEL
LIN {X 0,Y 148.265,Z 815.688,A -85,B 0,C 180,E1 25009.579,E2 25009.579} C_VEL
LIN {X 0,Y 156.883,Z 807.744,A -85,B 0,C 180,E1 25020.767,E2 25020.767} C_VEL
LIN {X 0,Y 157.878,Z 810.54,A -85,B 0,C 180,E1 25031.733,E2 25031.733} C_VEL
LIN {X 0,Y 154.857,Z 817.06,A -85,B 0,C 180,E1 25037.492,E2 25037.492} C_VEL
LIN {X 0,Y 148.086,Z 823.186,A -85,B 0,C 180,E1 25038.902,E2 25038.902} C_VEL
LIN {X 0,Y 118.976,Z 841.457,A -85,B 0,C 180,E1 25042.649,E2 25042.649} C_VEL
LIN {X 0,Y 83.273,Z 858.275,A -85,B 0,C 180,E1 25063.201,E2 25063.201} C_VEL
LIN {X 0,Y 70.506,Z 861.639,A -85,B 0,C 180,E1 25103.822,E2 25103.822} C_VEL
LIN {X 0,Y 70.875,Z 854.765,A -85,B 0,C 180,E1 25128.734,E2 25128.734} C_VEL
LIN {X 0,Y 87.772,Z 830.434,A -85,B 0,C 180,E1 25161.081,E2 25161.081} C_VEL
LIN {X 0,Y 114.666,Z 793.15,A -85,B 0,C 180,E1 25176.835,E2 25176.835} C_VEL
LIN {X 0,Y 118.214,Z 777.003,A -85,B 0,C 180,E1 25183.594,E2 25183.594} C_VEL
LIN {X 0,Y 117.719,Z 753.304,A -85,B 0,C 180,E1 25198.146,E2 25198.146} C_VEL
LIN {X 0,Y 116.449,Z 745.36,A -85,B 0,C 180,E1 25207.857,E2 25207.857} C_VEL
LIN {X 0,Y 114.72,Z 748.533,A -85,B 0,C 180,E1 25224.831,E2 25224.831} C_VEL
LIN {X 0,Y 115.244,Z 763.417,A -85,B 0,C 180,E1 25240.945,E2 25240.945} C_VEL
LIN {X 0,Y 111.778,Z 785.228,A -85,B 0,C 180,E1 25254.574,E2 25254.574} C_VEL
LIN {X 0,Y 87.056,Z 818.067,A -85,B 0,C 180,E1 25272.038,E2 25272.038} C_VEL
LIN {X 0,Y 72.663,Z 837.086,A -85,B 0,C 180,E1 25302.055,E2 25302.055} C_VEL
LIN {X 0,Y 78.71,Z 843.363,A -85,B 0,C 180,E1 25332.44,E2 25332.44} C_VEL
LIN {X 0,Y 106.564,Z 838.228,A -85,B 0,C 180,E1 25357.767,E2 25357.767} C_VEL
LIN {X 0,Y 141.947,Z 819.772,A -85,B 0,C 180,E1 25370.778,E2 25370.778} C_VEL
LIN {X 0,Y 151.911,Z 812.304,A -85,B 0,C 180,E1 25382.869,E2 25382.869} C_VEL
LIN {X 0,Y 151.295,Z 816.825,A -85,B 0,C 180,E1 25393.05,E2 25393.05} C_VEL
LIN {X 0,Y 147.641,Z 821.097,A -85,B 0,C 180,E1 25395.502,E2 25395.502} C_VEL
LIN {X 0,Y 118.976,Z 841.457,A -85,B 0,C 180,E1 25402.649,E2 25402.649} C_VEL
LIN {X 0,Y 88.709,Z 853.506,A -85,B 0,C 180,E1 25410.504,E2 25410.504} C_VEL
LIN {X 0,Y 62.779,Z 860.925,A -85,B 0,C 180,E1 25448.74,E2 25448.74} C_VEL
LIN {X 0,Y 62.785,Z 857.761,A -85,B 0,C 180,E1 25476.941,E2 25476.941} C_VEL
LIN {X 0,Y 73.548,Z 838.514,A -85,B 0,C 180,E1 25516.233,E2 25516.233} C_VEL
LIN {X 0,Y 101.231,Z 805.37,A -85,B 0,C 180,E1 25536.662,E2 25536.662} C_VEL
LIN {X 0,Y 111.461,Z 788.594,A -85,B 0,C 180,E1 25541.644,E2 25541.644} C_VEL
LIN {X 0,Y 113.7,Z 763.85,A -85,B 0,C 180,E1 25556.166,E2 25556.166} C_VEL
LIN {X 0,Y 113.19,Z 752.702,A -85,B 0,C 180,E1 25568.085,E2 25568.085} C_VEL
LIN {X 0,Y 111.118,Z 756.05,A -85,B 0,C 180,E1 25584.898,E2 25584.898} C_VEL
LIN {X 0,Y 110.163,Z 770.655,A -85,B 0,C 180,E1 25600.743,E2 25600.743} C_VEL
LIN {X 0,Y 105.09,Z 788.841,A -85,B 0,C 180,E1 25612.141,E2 25612.141} C_VEL
LIN {X 0,Y 79.233,Z 820.31,A -85,B 0,C 180,E1 25630.198,E2 25630.198} C_VEL
LIN {X 0,Y 64.526,Z 838.738,A -85,B 0,C 180,E1 25663.571,E2 25663.571} C_VEL
LIN {X 0,Y 72.719,Z 844.625,A -85,B 0,C 180,E1 25696.921,E2 25696.921} C_VEL
LIN {X 0,Y 103.659,Z 839.025,A -85,B 0,C 180,E1 25722.1,E2 25722.1} C_VEL
LIN {X 0,Y 137.138,Z 822.652,A -85,B 0,C 180,E1 25733.336,E2 25733.336} C_VEL
LIN {X 0,Y 145.431,Z 817.469,A -85,B 0,C 180,E1 25742.997,E2 25742.997} C_VEL
LIN {X 0,Y 145.273,Z 820.295,A -85,B 0,C 180,E1 25750.948,E2 25750.948} C_VEL
LIN {X 0,Y 140.312,Z 824.933,A -85,B 0,C 180,E1 25753.35,E2 25753.35} C_VEL
LIN {X 0,Y 100.167,Z 848.816,A -85,B 0,C 180,E1 25764.63,E2 25764.63} C_VEL
LIN {X 0,Y 88.709,Z 853.506,A -85,B 0,C 180,E1 25770.504,E2 25770.504} C_VEL
LIN {X 0,Y 61.596,Z 858.794,A -85,B 0,C 180,E1 25787.818,E2 25787.818} C_VEL
LIN {X 0,Y 54.999,Z 857.877,A -85,B 0,C 180,E1 25829.999,E2 25829.999} C_VEL
LIN {X 0,Y 63.098,Z 841.63,A -85,B 0,C 180,E1 25874.529,E2 25874.529} C_VEL
LIN {X 0,Y 91.861,Z 810.675,A -85,B 0,C 180,E1 25898.318,E2 25898.318} C_VEL
LIN {X 0,Y 105.79,Z 790.724,A -85,B 0,C 180,E1 25904.538,E2 25904.538} C_VEL
LIN {X 0,Y 109.274,Z 768.184,A -85,B 0,C 180,E1 25918.997,E2 25918.997} C_VEL
LIN {X 0,Y 109.629,Z 760.049,A -85,B 0,C 180,E1 25927.949,E2 25927.949} C_VEL
LIN {X 0,Y 107.35,Z 762.413,A -85,B 0,C 180,E1 25943.24,E2 25943.24} C_VEL
LIN {X 0,Y 105.215,Z 775.293,A -85,B 0,C 180,E1 25958.453,E2 25958.453} C_VEL
LIN {X 0,Y 99.596,Z 790.972,A -85,B 0,C 180,E1 25968.922,E2 25968.922} C_VEL
LIN {X 0,Y 71.053,Z 823.042,A -85,B 0,C 180,E1 25988.538,E2 25988.538} C_VEL
LIN {X 0,Y 56.432,Z 841.378,A -85,B 0,C 180,E1 26029.783,E2 26029.783} C_VEL
LIN {X 0,Y 76.981,Z 845.386,A -85,B 0,C 180,E1 26072.512,E2 26072.512} C_VEL
LIN {X 0,Y 115.098,Z 834.557,A -85,B 0,C 180,E1 26091.442,E2 26091.442} C_VEL
LIN {X 0,Y 133.22,Z 825.105,A -85,B 0,C 180,E1 26096.741,E2 26096.741} C_VEL
LIN {X 0,Y 138.718,Z 822.323,A -85,B 0,C 180,E1 26103.142,E2 26103.142} C_VEL
LIN {X 0,Y 137.54,Z 825.355,A -85,B 0,C 180,E1 26110.264,E2 26110.264} C_VEL
LIN {X 0,Y 93.804,Z 849.279,A -85,B 0,C 180,E1 26121.529,E2 26121.529} C_VEL
LIN {X 0,Y 61.596,Z 858.794,A -85,B 0,C 180,E1 26147.818,E2 26147.818} C_VEL
LIN {X 0,Y 46.546,Z 857.229,A -85,B 0,C 180,E1 26182.705,E2 26182.705} C_VEL
LIN {X 0,Y 48.159,Z 849.719,A -85,B 0,C 180,E1 26218.207,E2 26218.207} C_VEL
LIN {X 0,Y 73.22,Z 825.055,A -85,B 0,C 180,E1 26255.059,E2 26255.059} C_VEL
LIN {X 0,Y 100.699,Z 791.593,A -85,B 0,C 180,E1 26268.392,E2 26268.392} C_VEL
LIN {X 0,Y 105.115,Z 771.268,A -85,B 0,C 180,E1 26283.095,E2 26283.095} C_VEL
LIN {X 0,Y 105.022,Z 766.514,A -85,B 0,C 180,E1 26292.51,E2 26292.51} C_VEL
LIN {X 0,Y 102.052,Z 773.399,A -85,B 0,C 180,E1 26309.12,E2 26309.12} C_VEL
LIN {X 0,Y 96.783,Z 789.403,A -85,B 0,C 180,E1 26323.653,E2 26323.653} C_VEL
LIN {X 0,Y 67.803,Z 821.334,A -85,B 0,C 180,E1 26341.477,E2 26341.477} C_VEL
LIN {X 0,Y 48.549,Z 841.375,A -85,B 0,C 180,E1 26385.326,E2 26385.326} C_VEL
LIN {X 0,Y 62.432,Z 847.053,A -85,B 0,C 180,E1 26428.294,E2 26428.294} C_VEL
LIN {X 0,Y 99.768,Z 840.671,A -85,B 0,C 180,E1 26451.378,E2 26451.378} C_VEL
LIN {X 0,Y 125.674,Z 829.623,A -85,B 0,C 180,E1 26458.195,E2 26458.195} C_VEL
LIN {X 0,Y 131.714,Z 826.899,A -85,B 0,C 180,E1 26463.309,E2 26463.309} C_VEL
LIN {X 0,Y 130.179,Z 829.014,A -85,B 0,C 180,E1 26467.745,E2 26467.745} C_VEL
LIN {X 0,Y 84.428,Z 850.755,A -85,B 0,C 180,E1 26479.324,E2 26479.324} C_VEL
LIN {X 0,Y 53.95,Z 857.981,A -85,B 0,C 180,E1 26505.313,E2 26505.313} C_VEL
LIN {X 0,Y 46.546,Z 857.229,A -85,B 0,C 180,E1 26542.705,E2 26542.705} C_VEL
LIN {X 0,Y 42.818,Z 853.165,A -85,B 0,C 180,E1 26563.999,E2 26563.999} C_VEL
LIN {X 0,Y 42.212,Z 846.72,A -85,B 0,C 180,E1 26587.815,E2 26587.815} C_VEL
LIN {X 0,Y 71.747,Z 821.086,A -85,B 0,C 180,E1 26622.138,E2 26622.138} C_VEL
LIN {X 0,Y 95.665,Z 793.358,A -85,B 0,C 180,E1 26632.133,E2 26632.133} C_VEL
LIN {X 0,Y 101.033,Z 775.374,A -85,B 0,C 180,E1 26646.676,E2 26646.676} C_VEL
LIN {X 0,Y 99.778,Z 774.261,A -85,B 0,C 180,E1 26657.705,E2 26657.705} C_VEL
LIN {X 0,Y 96.026,Z 782.973,A -85,B 0,C 180,E1 26671.864,E2 26671.864} C_VEL
LIN {X 0,Y 89.598,Z 795.141,A -85,B 0,C 180,E1 26681.272,E2 26681.272} C_VEL
LIN {X 0,Y 57.842,Z 825.93,A -85,B 0,C 180,E1 26700.533,E2 26700.533} C_VEL
LIN {X 0,Y 40.6,Z 843.389,A -85,B 0,C 180,E1 26750.913,E2 26750.913} C_VEL
LIN {X 0,Y 61.892,Z 848.209,A -85,B 0,C 180,E1 26798.435,E2 26798.435} C_VEL
LIN {X 0,Y 102.555,Z 840.209,A -85,B 0,C 180,E1 26817.23,E2 26817.23} C_VEL
LIN {X 0,Y 120.433,Z 832.806,A -85,B 0,C 180,E1 26821.112,E2 26821.112} C_VEL
LIN {X 0,Y 124.874,Z 831.087,A -85,B 0,C 180,E1 26824.18,E2 26824.18} C_VEL
LIN {X 0,Y 78.633,Z 850.847,A -85,B 0,C 180,E1 26835.211,E2 26835.211} C_VEL
LIN {X 0,Y 41.018,Z 857.031,A -85,B 0,C 180,E1 26876.291,E2 26876.291} C_VEL
LIN {X 0,Y 39.093,Z 854.934,A -85,B 0,C 180,E1 26910.327,E2 26910.327} C_VEL
LIN {X 0,Y 42.212,Z 846.72,A -85,B 0,C 180,E1 26947.815,E2 26947.815} C_VEL
LIN {X 0,Y 56.191,Z 830.056,A -85,B 0,C 180,E1 26981.314,E2 26981.314} C_VEL
LIN {X 0,Y 90.314,Z 796.687,A -85,B 0,C 180,E1 26995.17,E2 26995.17} C_VEL
LIN {X 0,Y 96.515,Z 781.055,A -85,B 0,C 180,E1 27008.639,E2 27008.639} C_VEL
LIN {X 0,Y 94.038,Z 782.605,A -85,B 0,C 180,E1 27021.617,E2 27021.617} C_VEL
LIN {X 0,Y 87.953,Z 793.838,A -85,B 0,C 180,E1 27035.27,E2 27035.27} C_VEL
LIN {X 0,Y 55.372,Z 824.639,A -85,B 0,C 180,E1 27051.929,E2 27051.929} C_VEL
LIN {X 0,Y 32.723,Z 843.116,A -85,B 0,C 180,E1 27103.409,E2 27103.409} C_VEL
LIN {X 0,Y 55.47,Z 849.484,A -85,B 0,C 180,E1 27163.242,E2 27163.242} C_VEL
LIN {X 0,Y 102.046,Z 841.133,A -85,B 0,C 180,E1 27181.853,E2 27181.853} C_VEL
LIN {X 0,Y 105.446,Z 839.943,A -85,B 0,C 180,E1 27182.528,E2 27182.528} C_VEL
LIN {X 0,Y 56.06,Z 854.168,A -85,B 0,C 180,E1 27198.656,E2 27198.656} C_VEL
LIN {X 0,Y 30.742,Z 854.627,A -85,B 0,C 180,E1 27255.71,E2 27255.71} C_VEL
LIN {X 0,Y 31.174,Z 850.419,A -85,B 0,C 180,E1 27291.412,E2 27291.412} C_VEL
LIN {X 0,Y 56.191,Z 830.056,A -85,B 0,C 180,E1 27341.314,E2 27341.314} C_VEL
LIN {X 0,Y 76.953,Z 808.18,A -85,B 0,C 180,E1 27357.631,E2 27357.631} C_VEL
LIN {X 0,Y 86.588,Z 797.203,A -85,B 0,C 180,E1 27360.562,E2 27360.562} C_VEL
LIN {X 0,Y 91.375,Z 787.544,A -85,B 0,C 180,E1 27369.551,E2 27369.551} C_VEL
LIN {X 0,Y 88.171,Z 790.189,A -85,B 0,C 180,E1 27383.047,E2 27383.047} C_VEL
LIN {X 0,Y 82.217,Z 798.489,A -85,B 0,C 180,E1 27391.841,E2 27391.841} C_VEL
LIN {X 0,Y 45.917,Z 829,A -85,B 0,C 180,E1 27408.625,E2 27408.625} C_VEL
LIN {X 0,Y 26.097,Z 846.836,A -85,B 0,C 180,E1 27487.205,E2 27487.205} C_VEL
LIN {X 0,Y 53.652,Z 850.668,A -85,B 0,C 180,E1 27531.886,E2 27531.886} C_VEL
LIN {X 0,Y 77.656,Z 848.299,A -85,B 0,C 180,E1 27541.412,E2 27541.412} C_VEL
LIN {X 0,Y 40.36,Z 854.296,A -85,B 0,C 180,E1 27559.943,E2 27559.943} C_VEL
LIN {X 0,Y 22.896,Z 851.455,A -85,B 0,C 180,E1 27635.782,E2 27635.782} C_VEL
LIN {X 0,Y 50.493,Z 830.514,A -85,B 0,C 180,E1 27707.625,E2 27707.625} C_VEL
LIN {X 0,Y 76.953,Z 808.18,A -85,B 0,C 180,E1 27717.631,E2 27717.631} C_VEL
LIN {X 0,Y 83.074,Z 799.057,A -85,B 0,C 180,E1 27724.588,E2 27724.588} C_VEL
LIN {X 0,Y 85.56,Z 794.352,A -85,B 0,C 180,E1 27730.101,E2 27730.101} C_VEL
LIN {X 0,Y 83.336,Z 795.587,A -85,B 0,C 180,E1 27740.762,E2 27740.762} C_VEL
LIN {X 0,Y 78.224,Z 801.449,A -85,B 0,C 180,E1 27746.763,E2 27746.763} C_VEL
LIN {X 0,Y 38.454,Z 832.091,A -85,B 0,C 180,E1 27762.274,E2 27762.274} C_VEL
LIN {X 0,Y 19.732,Z 848.218,A -85,B 0,C 180,E1 27860.275,E2 27860.275} C_VEL
LIN {X 0,Y 53.138,Z 851.922,A -85,B 0,C 180,E1 27901.691,E2 27901.691} C_VEL
LIN {X 0,Y 14.945,Z 850.835,A -85,B 0,C 180,E1 27983.628,E2 27983.628} C_VEL
LIN {X 0,Y 43.819,Z 831.917,A -85,B 0,C 180,E1 28074.663,E2 28074.663} C_VEL
LIN {X 0,Y 82.527,Z 799.356,A -85,B 0,C 180,E1 28085.265,E2 28085.265} C_VEL
LIN {X 0,Y 85.56,Z 794.352,A -85,B 0,C 180,E1 28090.101,E2 28090.101} C_VEL
LIN {X 0,Y 78.808,Z 800.516,A -85,B 0,C 180,E1 28096.993,E2 28096.993} C_VEL
LIN {X 0,Y 75.421,Z 803.779,A -85,B 0,C 180,E1 28101.128,E2 28101.128} C_VEL
LIN {X 0,Y 35.374,Z 833.089,A -85,B 0,C 180,E1 28110.908,E2 28110.908} C_VEL
LIN {X 0,Y 15.754,Z 849.701,A -85,B 0,C 180,E1 28244.429,E2 28244.429} C_VEL
LIN {X 0,Y 27.437,Z 851.784,A -85,B 0,C 180,E1 28259.869,E2 28259.869} C_VEL
LIN {X 0,Y 7.37,Z 847.923,A -85,B 0,C 180,E1 28380.978,E2 28380.978} C_VEL
LIN {X 0,Y 49.653,Z 826.039,A -85,B 0,C 180,E1 28446.644,E2 28446.644} C_VEL
LIN {X 0,Y 79.134,Z 801.14,A -85,B 0,C 180,E1 28450.761,E2 28450.761} C_VEL
LIN {X 0,Y 78.808,Z 800.516,A -85,B 0,C 180,E1 28456.993,E2 28456.993} C_VEL
LIN {X 0,Y 68.981,Z 809.753,A -85,B 0,C 180,E1 28461.249,E2 28461.249} C_VEL
LIN {X 0,Y 45.394,Z 827.55,A -85,B 0,C 180,E1 28456.844,E2 28456.844} C_VEL
LIN {X 0,Y 8.106,Z 845.035,A -85,B 0,C 180,E1 28460.607,E2 28460.607} C_VEL
LIN {X 0,Y 53.003,Z 822.618,A -85,B 0,C 180,E1 28455.854,E2 28455.854} C_VEL
LIN {X 0,Y 55.35,Z 820.872,A -85,B 0,C 180,E1 28456.344,E2 28456.344} C_VEL
LIN {X 0,Y 45.394,Z 827.55,A -85,B 0,C 180,E1 28456.844,E2 28456.844} C_VEL
LIN {X 0,Y 44.42,Z 829.267,A -85,B 0,C 180,E1 28456.897,E2 28456.897} C_VEL
LIN {X 0,Y 44.42,Z 931,A -85,B 0,C 180,E1 28456.897,E2 28456.897} C_VEL
LIN {X 0,Y 44.42,Z 931,A -85,B 0,C 180,E1 28456.897,E2 28456.897}

